SUBAPPLICATION Uebung_016a (* Background Colour umschalten -- 3-fach *)
  (* Standard: 61499-2; Description: Copyright (c) 2023 Meisterschulen am Ostbahnhof This program and the accompanying materials are made available under the terms of the Eclipse Public License 2.0 which is available at https://www.eclipse.org/legal/epl-2.0/ SPDX-License-Identifier: EPL-2.0 *)
  (* Version 1.0, 2023-10-23, Franz Höpfinger, Meisterschulen am Ostbahnhof *)
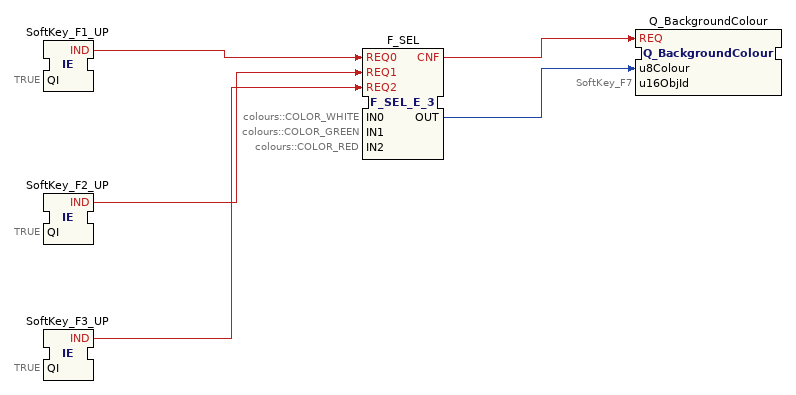
  FBS
    SoftKey_F1_UP : IE(QI := TRUE);
    SoftKey_F2_UP : IE(QI := TRUE);
    F_SEL : F_SEL_E_3(IN0 := colours::COLOR_WHITE, IN1 := colours::COLOR_GREEN, IN2 := colours::COLOR_RED);
    Q_BackgroundColour : Q_BackgroundColour(u16ObjId := SoftKey_F7);
    SoftKey_F3_UP : IE(QI := TRUE);
  END_FBS
  EVENT_CONNECTIONS
    F_SEL.CNF TO Q_BackgroundColour.REQ;
    SoftKey_F1_UP.IND TO F_SEL.REQ0;
    SoftKey_F2_UP.IND TO F_SEL.REQ1;
    SoftKey_F3_UP.IND TO F_SEL.REQ2;
  END_CONNECTIONS
  DATA_CONNECTIONS
    F_SEL.OUT TO Q_BackgroundColour.u8Colour;
  END_CONNECTIONS
END_SUBAPPLICATION
